// TIA Portal project "Traffic Contol" (V14)

(* hardware
DEVICE "S7-1200 station_1"  S7-1200 Station
   slot 0: "Rack_0"  S7-1200 Rack  Rack  V1.0
   slot 1: "PLC_1"  CPU 1212C AC/DC/Rly  6ES7 212-1BE40-0XB0  V4.2
DEVICE "S7-1200 station_2"  S7-1200 Station
   slot 0: "Rack_0"  S7-1200 Rack  Rack  V1.0
   slot 1: "PLC_2"  CPU 1212C AC/DC/Rly  6ES7 212-1BE40-0XB0  V4.2
*)

// ===== PLC "PLC_1"  CPU 1212C AC/DC/Rly =====

VAR_GLOBAL   // PLC tag table "Default tag table"
   "Switch_0" AT %I0.0 : Bool;
   "Switch_1" AT %I0.1 : Bool;
   "Switch_2" AT %I0.2 : Bool;
   "Switch_3" AT %I0.3 : Bool;
   "Switch_4" AT %I0.4 : Bool;
   "Switch_5" AT %I0.5 : Bool;
   "Switch_6" AT %I0.6 : Bool;
   "Switch_7" AT %I0.7 : Bool;
   "Green_light_1" AT %Q0.0 : Bool;
   "Yellow_light_1" AT %Q0.1 : Bool;
   "Red_light_1" AT %Q0.2 : Bool;
   "Yellow_light_2" AT %Q0.3 : Bool;
   "Red_light_2" AT %Q0.4 : Bool;
   "Green_light_2" AT %Q0.5 : Bool;
   "Delay_1" AT %M0.0 : Bool;
   "Delay_2" AT %M0.1 : Bool;
   "System_Byte" AT %MB1 : Byte;
   "FirstScan" AT %M1.0 : Bool;
   "DiagStatusUpdate" AT %M1.1 : Bool;
   "AlwaysTRUE" AT %M1.2 : Bool;
   "AlwaysFALSE" AT %M1.3 : Bool;
   "System_Byte(1)" AT %MB1 : Byte;
   "Clock_Byte" AT %MB5 : Byte;
   "Clock_10Hz" AT %M5.0 : Bool;
   "Clock_5Hz" AT %M5.1 : Bool;
   "Clock_2.5Hz" AT %M5.2 : Bool;
   "Clock_2Hz" AT %M5.3 : Bool;
   "Clock_1.25Hz" AT %M5.4 : Bool;
   "Clock_1Hz" AT %M5.5 : Bool;
   "Clock_0.625Hz" AT %M5.6 : Bool;
   "Clock_0.5Hz" AT %M5.7 : Bool;
   "ERR" AT %MW2 : Int;
END_VAR

DATA_BLOCK "HOLD_REG"   // DB10
{ S7_Optimized_Access := 'FALSE' }
VERSION : 0.1
   VAR
      BUFFER : Array[0..15] of Bool;
      BUFFER1 : Array[0..15] of Bool;
      FILLER : Array[0..15] of Word;
   END_VAR
BEGIN
   BUFFER[2] := false;
   BUFFER[0] := false;
   BUFFER[6] := false;
END_DATA_BLOCK

DATA_BLOCK "CONFIG_PLC_2"   // DB11
{ S7_Optimized_Access := 'TRUE' }
VERSION : 0.1
   VAR
      Server_IP : TCON_IP_v4;
      DISCONNECT : Bool;
      NDR : Bool;
      DR : Bool;
      ERROR : Bool;
      STATUS : Word;
   END_VAR
BEGIN
   Server_IP.InterfaceId := 64;
   Server_IP.LocalPort := 502;
   Server_IP.ID := 16#01;
END_DATA_BLOCK

DATA_BLOCK "CONFIG_Train"   // DB14
{ S7_Optimized_Access := 'TRUE' }
VERSION : 0.1
   VAR
      Server_IP : TCON_IP_v4;
      DISCONNECT : Bool;
      NDR : Bool;
      DR : Bool;
      ERROR : Bool;
      STATUS : Word;
   END_VAR
BEGIN
   Server_IP.InterfaceId := 64;
   Server_IP.LocalPort := 503;
   Server_IP.ID := 16#03;
END_DATA_BLOCK

DATA_BLOCK "CONFIG_Overide"   // DB15
{ S7_Optimized_Access := 'TRUE' }
VERSION : 0.1
   VAR
      Server_IP : TCON_IP_v4;
      DISCONNECT : Bool := false;
      NDR : Bool := false;
      DR : Bool := false;
      ERROR : Bool := false;
      STATUS : Word := 16#0;
   END_VAR
BEGIN
   Server_IP.InterfaceId := 64;
   Server_IP.LocalPort := 504;
   Server_IP.ID := 16#04;
END_DATA_BLOCK

// folder: System blocks/Program resources

DATA_BLOCK "IEC_Timer_0_DB"   // DB1
{ S7_Optimized_Access := 'TRUE' }
AUTHOR : Simatic
FAMILY : IEC
NAME : IEC_TMR
VERSION : 1.0
// stored: InstanceOfName IEC_TIMER
"IEC_TIMER"
BEGIN
END_DATA_BLOCK

DATA_BLOCK "IEC_Timer_0_DB_1"   // DB2
{ S7_Optimized_Access := 'TRUE' }
AUTHOR : Simatic
FAMILY : IEC
NAME : IEC_TMR
VERSION : 1.0
// stored: InstanceOfName IEC_TIMER
"IEC_TIMER"
BEGIN
END_DATA_BLOCK

DATA_BLOCK "IEC_Timer_0_DB_2"   // DB3
{ S7_Optimized_Access := 'TRUE' }
AUTHOR : Simatic
FAMILY : IEC
NAME : IEC_TMR
VERSION : 1.0
// stored: InstanceOfName IEC_TIMER
"IEC_TIMER"
BEGIN
END_DATA_BLOCK

DATA_BLOCK "IEC_Timer_0_DB_3"   // DB4
{ S7_Optimized_Access := 'TRUE' }
AUTHOR : Simatic
FAMILY : IEC
NAME : IEC_TMR
VERSION : 1.0
// stored: InstanceOfName IEC_TIMER
"IEC_TIMER"
BEGIN
END_DATA_BLOCK

DATA_BLOCK "IEC_Timer_0_DB_4"   // DB5
{ S7_Optimized_Access := 'TRUE' }
AUTHOR : Simatic
FAMILY : IEC
NAME : IEC_TMR
VERSION : 1.0
// stored: InstanceOfName IEC_TIMER
"IEC_TIMER"
BEGIN
END_DATA_BLOCK

DATA_BLOCK "IEC_Timer_0_DB_5"   // DB6
{ S7_Optimized_Access := 'TRUE' }
AUTHOR : Simatic
FAMILY : IEC
NAME : IEC_TMR
VERSION : 1.0
// stored: InstanceOfName IEC_TIMER
"IEC_TIMER"
BEGIN
END_DATA_BLOCK

DATA_BLOCK "IEC_Timer_0_DB_6"   // DB7
{ S7_Optimized_Access := 'TRUE' }
AUTHOR : Simatic
FAMILY : IEC
NAME : IEC_TMR
VERSION : 1.0
// stored: InstanceOfName IEC_TIMER
"IEC_TIMER"
BEGIN
END_DATA_BLOCK

DATA_BLOCK "IEC_Timer_0_DB_7"   // DB8
{ S7_Optimized_Access := 'TRUE' }
AUTHOR : Simatic
FAMILY : IEC
NAME : IEC_TMR
VERSION : 1.0
// stored: InstanceOfName IEC_TIMER
"IEC_TIMER"
BEGIN
END_DATA_BLOCK

DATA_BLOCK "IEC_Timer_0_DB_8"   // DB9
{ S7_Optimized_Access := 'TRUE' }
AUTHOR : Simatic
FAMILY : IEC
NAME : IEC_TMR
VERSION : 1.0
// stored: InstanceOfName IEC_TIMER
"IEC_TIMER"
BEGIN
END_DATA_BLOCK

// folder: (top level)

FUNCTION "Trash" : Void   // FC1, LAD
{ S7_Optimized_Access := 'TRUE' }
VERSION : 0.1
   VAR_TEMP   // added for the SCL form of the ladder/FBD networks
      _w1 : Bool;
   END_VAR
BEGIN

REGION Network 2
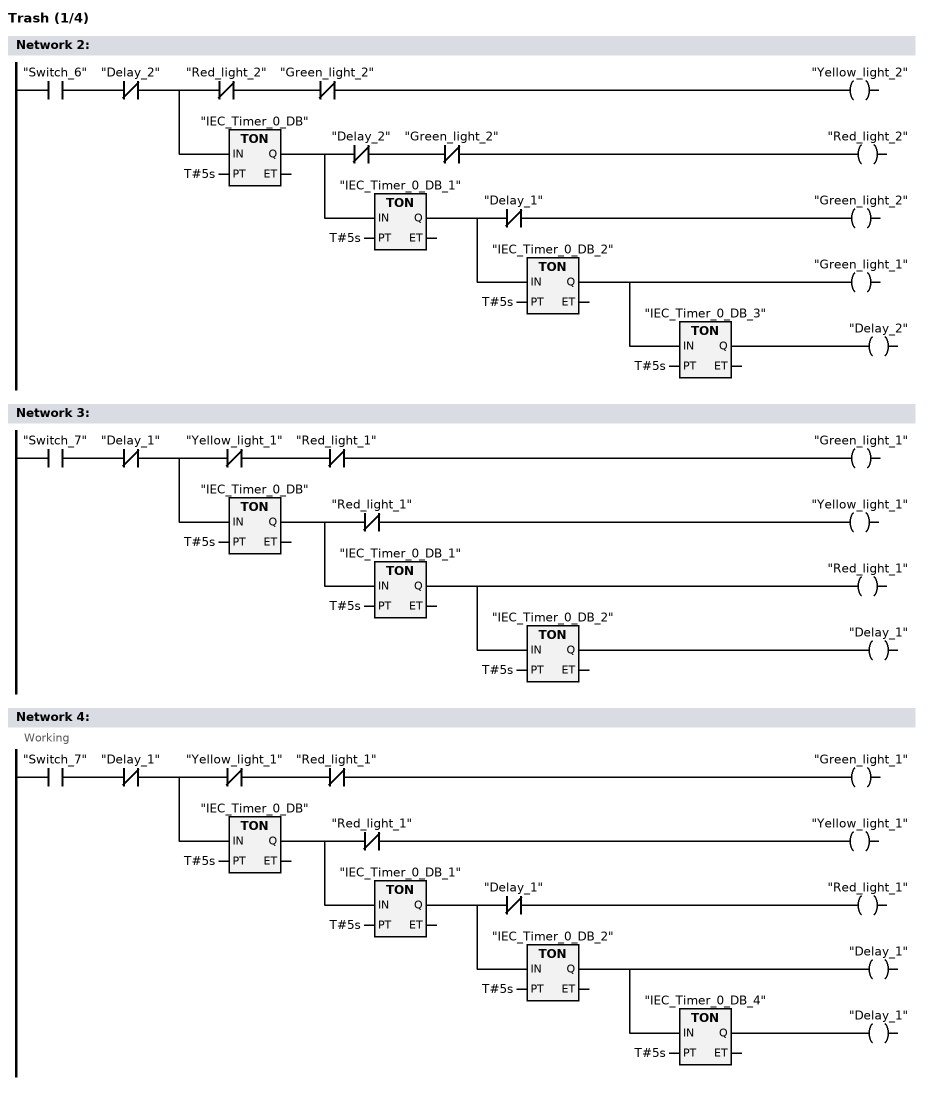
   #_w1 := "Switch_6" AND NOT "Delay_2";
   "Yellow_light_2" := #_w1 AND NOT "Red_light_2" AND NOT "Green_light_2";
   "IEC_Timer_0_DB".TON(IN := #_w1, PT := T#5s);
   "Red_light_2" := "IEC_Timer_0_DB".Q AND NOT "Delay_2" AND NOT "Green_light_2";
   "IEC_Timer_0_DB_1".TON(IN := "IEC_Timer_0_DB".Q, PT := T#5s);
   "Green_light_2" := "IEC_Timer_0_DB_1".Q AND NOT "Delay_1";
   "IEC_Timer_0_DB_2".TON(IN := "IEC_Timer_0_DB_1".Q, PT := T#5s);
   "Green_light_1" := "IEC_Timer_0_DB_2".Q;
   "IEC_Timer_0_DB_3".TON(IN := "IEC_Timer_0_DB_2".Q, PT := T#5s);
   "Delay_2" := "IEC_Timer_0_DB_3".Q;
END_REGION

REGION Network 3
   #_w1 := "Switch_7" AND NOT "Delay_1";
   "Green_light_1" := #_w1 AND NOT "Yellow_light_1" AND NOT "Red_light_1";
   "IEC_Timer_0_DB".TON(IN := #_w1, PT := T#5s);
   "Yellow_light_1" := "IEC_Timer_0_DB".Q AND NOT "Red_light_1";
   "IEC_Timer_0_DB_1".TON(IN := "IEC_Timer_0_DB".Q, PT := T#5s);
   "Red_light_1" := "IEC_Timer_0_DB_1".Q;
   "IEC_Timer_0_DB_2".TON(IN := "IEC_Timer_0_DB_1".Q, PT := T#5s);
   "Delay_1" := "IEC_Timer_0_DB_2".Q;
END_REGION

REGION Network 4
   // Working
   #_w1 := "Switch_7" AND NOT "Delay_1";
   "Green_light_1" := #_w1 AND NOT "Yellow_light_1" AND NOT "Red_light_1";
   "IEC_Timer_0_DB".TON(IN := #_w1, PT := T#5s);
   "Yellow_light_1" := "IEC_Timer_0_DB".Q AND NOT "Red_light_1";
   "IEC_Timer_0_DB_1".TON(IN := "IEC_Timer_0_DB".Q, PT := T#5s);
   "Red_light_1" := "IEC_Timer_0_DB_1".Q AND NOT "Delay_1";
   "IEC_Timer_0_DB_2".TON(IN := "IEC_Timer_0_DB_1".Q, PT := T#5s);
   "Delay_1" := "IEC_Timer_0_DB_2".Q;
   "IEC_Timer_0_DB_4".TON(IN := "IEC_Timer_0_DB_2".Q, PT := T#5s);
   "Delay_1" := "IEC_Timer_0_DB_4".Q;
END_REGION

REGION Network 5
   // Working 123
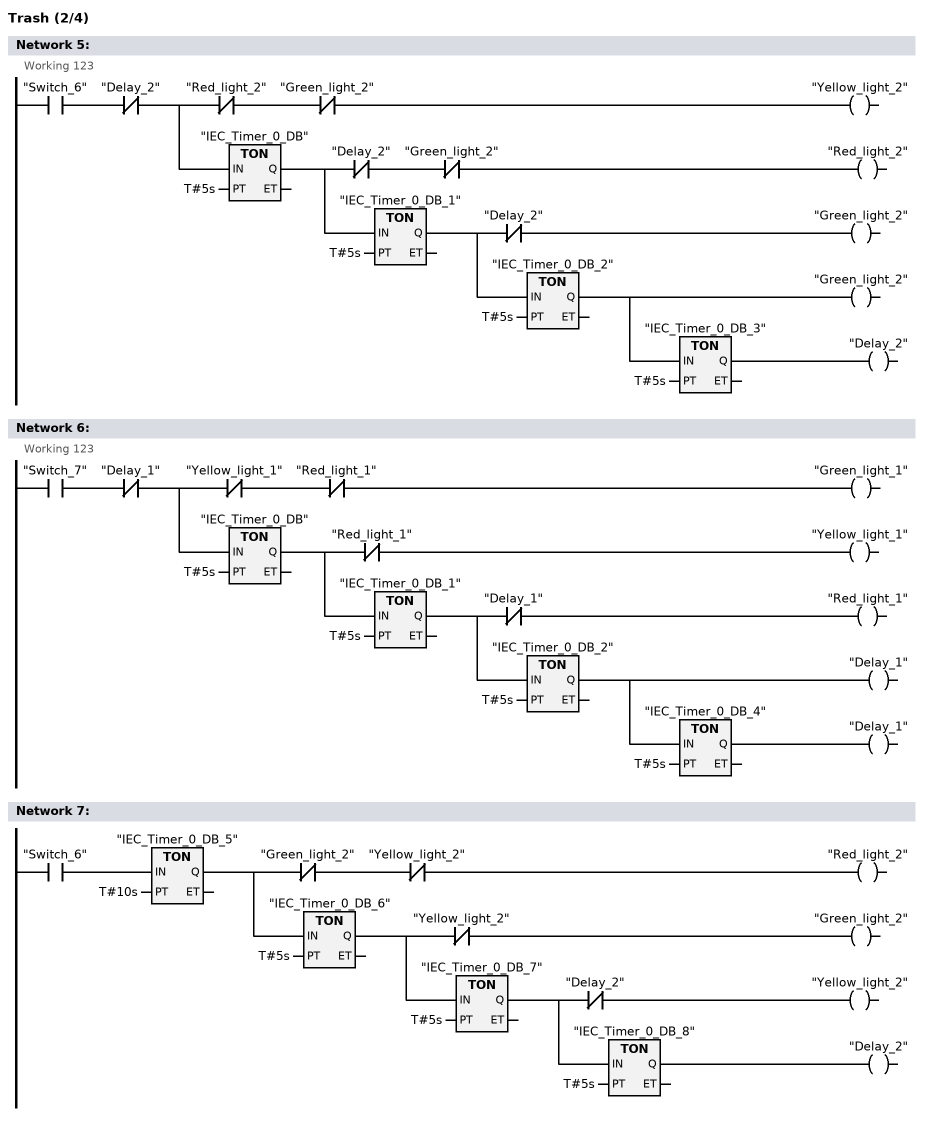
   #_w1 := "Switch_6" AND NOT "Delay_2";
   "Yellow_light_2" := #_w1 AND NOT "Red_light_2" AND NOT "Green_light_2";
   "IEC_Timer_0_DB".TON(IN := #_w1, PT := T#5s);
   "Red_light_2" := "IEC_Timer_0_DB".Q AND NOT "Delay_2" AND NOT "Green_light_2";
   "IEC_Timer_0_DB_1".TON(IN := "IEC_Timer_0_DB".Q, PT := T#5s);
   "Green_light_2" := "IEC_Timer_0_DB_1".Q AND NOT "Delay_2";
   "IEC_Timer_0_DB_2".TON(IN := "IEC_Timer_0_DB_1".Q, PT := T#5s);
   "Green_light_2" := "IEC_Timer_0_DB_2".Q;
   "IEC_Timer_0_DB_3".TON(IN := "IEC_Timer_0_DB_2".Q, PT := T#5s);
   "Delay_2" := "IEC_Timer_0_DB_3".Q;
END_REGION

REGION Network 6
   // Working 123
   #_w1 := "Switch_7" AND NOT "Delay_1";
   "Green_light_1" := #_w1 AND NOT "Yellow_light_1" AND NOT "Red_light_1";
   "IEC_Timer_0_DB".TON(IN := #_w1, PT := T#5s);
   "Yellow_light_1" := "IEC_Timer_0_DB".Q AND NOT "Red_light_1";
   "IEC_Timer_0_DB_1".TON(IN := "IEC_Timer_0_DB".Q, PT := T#5s);
   "Red_light_1" := "IEC_Timer_0_DB_1".Q AND NOT "Delay_1";
   "IEC_Timer_0_DB_2".TON(IN := "IEC_Timer_0_DB_1".Q, PT := T#5s);
   "Delay_1" := "IEC_Timer_0_DB_2".Q;
   "IEC_Timer_0_DB_4".TON(IN := "IEC_Timer_0_DB_2".Q, PT := T#5s);
   "Delay_1" := "IEC_Timer_0_DB_4".Q;
END_REGION

REGION Network 7
   "IEC_Timer_0_DB_5".TON(IN := "Switch_6", PT := T#10s);
   "Red_light_2" := "IEC_Timer_0_DB_5".Q AND NOT "Green_light_2" AND NOT "Yellow_light_2";
   "IEC_Timer_0_DB_6".TON(IN := "IEC_Timer_0_DB_5".Q, PT := T#5s);
   "Green_light_2" := "IEC_Timer_0_DB_6".Q AND NOT "Yellow_light_2";
   "IEC_Timer_0_DB_7".TON(IN := "IEC_Timer_0_DB_6".Q, PT := T#5s);
   "Yellow_light_2" := "IEC_Timer_0_DB_7".Q AND NOT "Delay_2";
   "IEC_Timer_0_DB_8".TON(IN := "IEC_Timer_0_DB_7".Q, PT := T#5s);
   "Delay_2" := "IEC_Timer_0_DB_8".Q;
END_REGION

REGION Network 8
   // working set
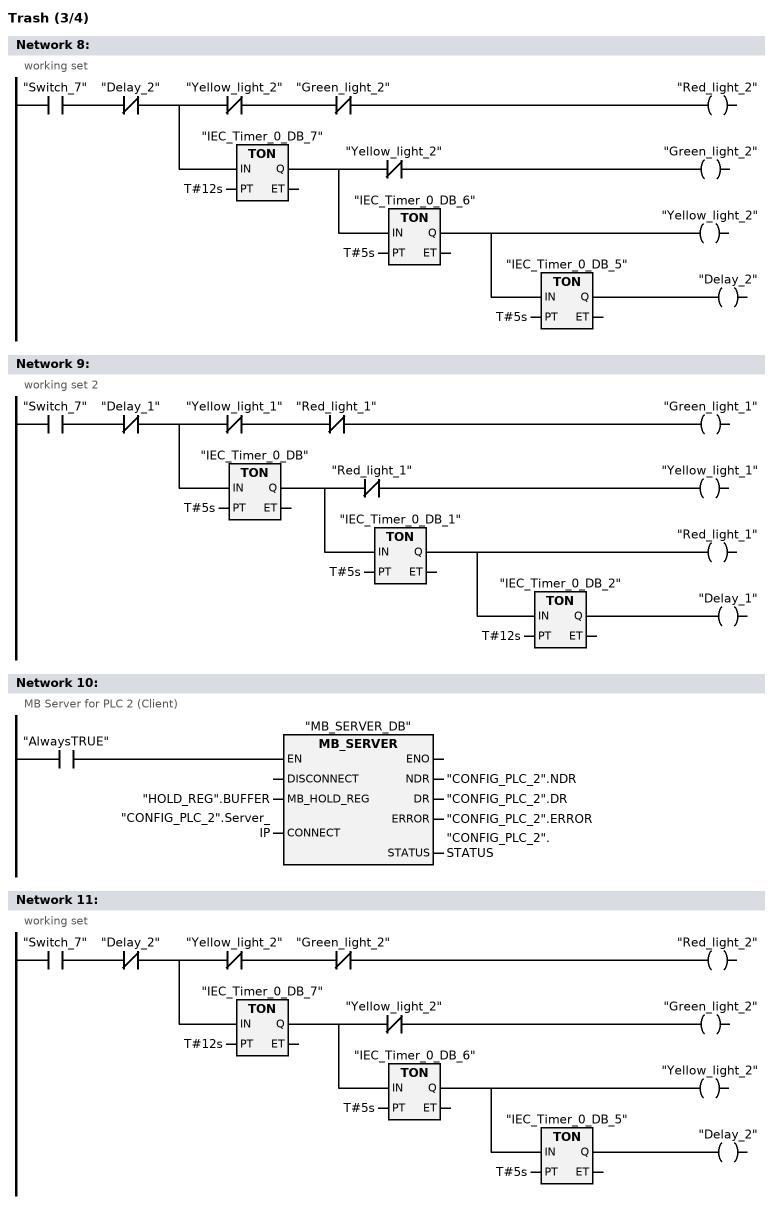
   #_w1 := "Switch_7" AND NOT "Delay_2";
   "Red_light_2" := #_w1 AND NOT "Yellow_light_2" AND NOT "Green_light_2";
   "IEC_Timer_0_DB_7".TON(IN := #_w1, PT := T#12s);
   "Green_light_2" := "IEC_Timer_0_DB_7".Q AND NOT "Yellow_light_2";
   "IEC_Timer_0_DB_6".TON(IN := "IEC_Timer_0_DB_7".Q, PT := T#5s);
   "Yellow_light_2" := "IEC_Timer_0_DB_6".Q;
   "IEC_Timer_0_DB_5".TON(IN := "IEC_Timer_0_DB_6".Q, PT := T#5s);
   "Delay_2" := "IEC_Timer_0_DB_5".Q;
END_REGION

REGION Network 9
   // working set 2
   #_w1 := "Switch_7" AND NOT "Delay_1";
   "Green_light_1" := #_w1 AND NOT "Yellow_light_1" AND NOT "Red_light_1";
   "IEC_Timer_0_DB".TON(IN := #_w1, PT := T#5s);
   "Yellow_light_1" := "IEC_Timer_0_DB".Q AND NOT "Red_light_1";
   "IEC_Timer_0_DB_1".TON(IN := "IEC_Timer_0_DB".Q, PT := T#5s);
   "Red_light_1" := "IEC_Timer_0_DB_1".Q;
   "IEC_Timer_0_DB_2".TON(IN := "IEC_Timer_0_DB_1".Q, PT := T#12s);
   "Delay_1" := "IEC_Timer_0_DB_2".Q;
END_REGION

REGION Network 10
   // MB Server for PLC 2 (Client)
   IF "AlwaysTRUE" THEN
       "MB_SERVER_DB"(MB_HOLD_REG := "HOLD_REG".BUFFER,   // MB_SERVER
                      CONNECT := "CONFIG_PLC_2".Server_IP,
                      NDR => "CONFIG_PLC_2".NDR,
                      DR => "CONFIG_PLC_2".DR,
                      ERROR => "CONFIG_PLC_2".ERROR,
                      STATUS => "CONFIG_PLC_2".STATUS);
   END_IF;
END_REGION

REGION Network 11
   // working set
   #_w1 := "Switch_7" AND NOT "Delay_2";
   "Red_light_2" := #_w1 AND NOT "Yellow_light_2" AND NOT "Green_light_2";
   "IEC_Timer_0_DB_7".TON(IN := #_w1, PT := T#12s);
   "Green_light_2" := "IEC_Timer_0_DB_7".Q AND NOT "Yellow_light_2";
   "IEC_Timer_0_DB_6".TON(IN := "IEC_Timer_0_DB_7".Q, PT := T#5s);
   "Yellow_light_2" := "IEC_Timer_0_DB_6".Q;
   "IEC_Timer_0_DB_5".TON(IN := "IEC_Timer_0_DB_6".Q, PT := T#5s);
   "Delay_2" := "IEC_Timer_0_DB_5".Q;
END_REGION

REGION Network 12
   // working set 2
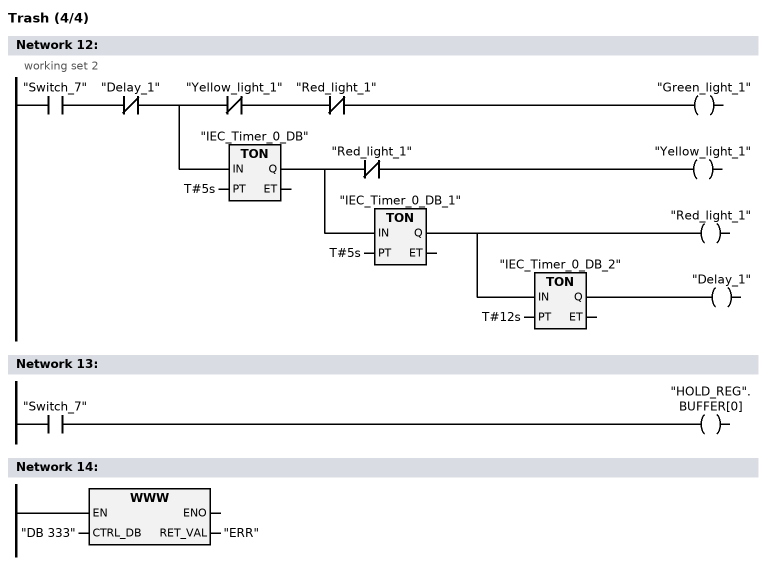
   #_w1 := "Switch_7" AND NOT "Delay_1";
   "Green_light_1" := #_w1 AND NOT "Yellow_light_1" AND NOT "Red_light_1";
   "IEC_Timer_0_DB".TON(IN := #_w1, PT := T#5s);
   "Yellow_light_1" := "IEC_Timer_0_DB".Q AND NOT "Red_light_1";
   "IEC_Timer_0_DB_1".TON(IN := "IEC_Timer_0_DB".Q, PT := T#5s);
   "Red_light_1" := "IEC_Timer_0_DB_1".Q;
   "IEC_Timer_0_DB_2".TON(IN := "IEC_Timer_0_DB_1".Q, PT := T#12s);
   "Delay_1" := "IEC_Timer_0_DB_2".Q;
END_REGION

REGION Network 13
   RUNG wire#powerrail
      Contact( "Switch_7" )
      Coil( "HOLD_REG".BUFFER[0] )
   END_RUNG
   // the same network as SCL:
   "HOLD_REG".BUFFER[0] := "Switch_7";
END_REGION

REGION Network 14
   "ERR" := WWW(CTRL_DB := "DB 333");
END_REGION
END_FUNCTION

ORGANIZATION_BLOCK "Main"   // OB1, LAD, ProgramCycle
TITLE = "Main Program Sweep (Cycle)"
{ S7_Optimized_Access := 'TRUE' }
VERSION : 0.1
   VAR_INPUT
      Initial_Call : Bool;   // Initial call of this OB
      Remanence : Bool;   // =True, if remanent data are available
   END_VAR
   VAR_TEMP   // added for the SCL form of the ladder/FBD networks
      _w1 : Bool;
   END_VAR
BEGIN

REGION Network 1
   // MB Server for overide
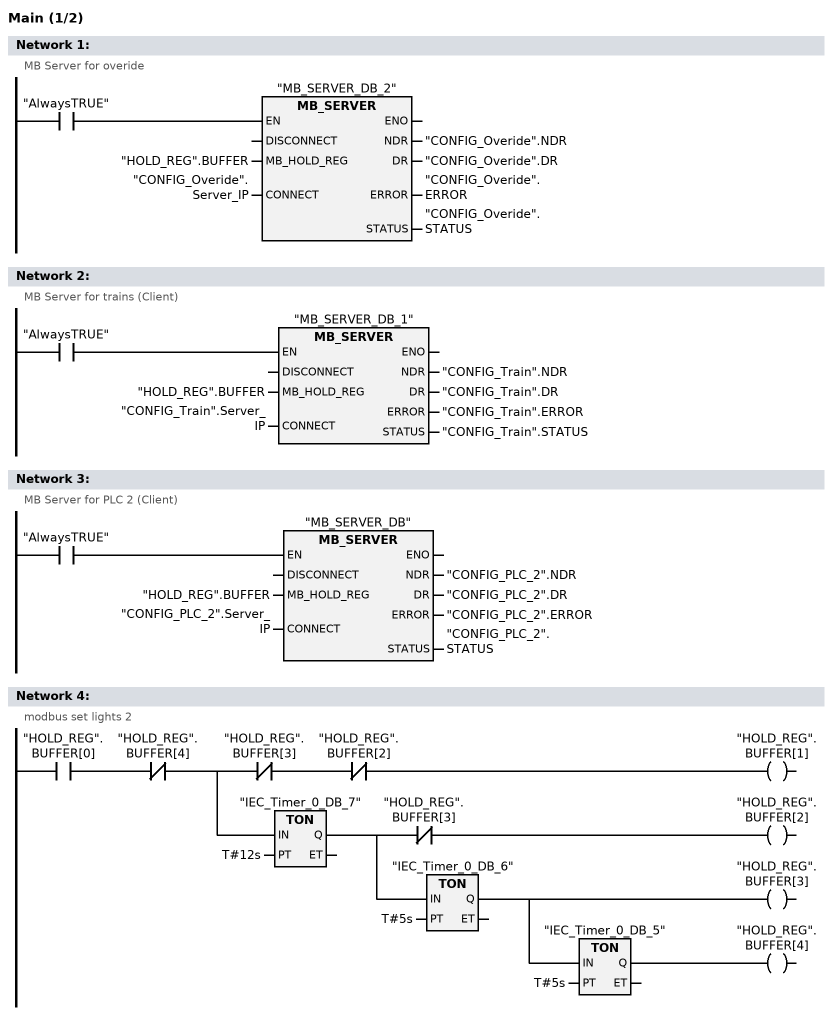
   IF "AlwaysTRUE" THEN
       "MB_SERVER_DB_2"(MB_HOLD_REG := "HOLD_REG".BUFFER,   // MB_SERVER
                        CONNECT := "CONFIG_Overide".Server_IP,
                        NDR => "CONFIG_Overide".NDR,
                        DR => "CONFIG_Overide".DR,
                        ERROR => "CONFIG_Overide".ERROR,
                        STATUS => "CONFIG_Overide".STATUS);
   END_IF;
END_REGION

REGION Network 2
   // MB Server for trains (Client)
   IF "AlwaysTRUE" THEN
       "MB_SERVER_DB_1"(MB_HOLD_REG := "HOLD_REG".BUFFER,   // MB_SERVER
                        CONNECT := "CONFIG_Train".Server_IP,
                        NDR => "CONFIG_Train".NDR,
                        DR => "CONFIG_Train".DR,
                        ERROR => "CONFIG_Train".ERROR,
                        STATUS => "CONFIG_Train".STATUS);
   END_IF;
END_REGION

REGION Network 3
   // MB Server for PLC 2 (Client)
   IF "AlwaysTRUE" THEN
       "MB_SERVER_DB"(MB_HOLD_REG := "HOLD_REG".BUFFER,   // MB_SERVER
                      CONNECT := "CONFIG_PLC_2".Server_IP,
                      NDR => "CONFIG_PLC_2".NDR,
                      DR => "CONFIG_PLC_2".DR,
                      ERROR => "CONFIG_PLC_2".ERROR,
                      STATUS => "CONFIG_PLC_2".STATUS);
   END_IF;
END_REGION

REGION Network 4
   // modbus set lights 2
   #_w1 := "HOLD_REG".BUFFER[0] AND NOT "HOLD_REG".BUFFER[4];
   "HOLD_REG".BUFFER[1] := #_w1 AND NOT "HOLD_REG".BUFFER[3] AND NOT "HOLD_REG".BUFFER[2];
   "IEC_Timer_0_DB_7".TON(IN := #_w1, PT := T#12s);
   "HOLD_REG".BUFFER[2] := "IEC_Timer_0_DB_7".Q AND NOT "HOLD_REG".BUFFER[3];
   "IEC_Timer_0_DB_6".TON(IN := "IEC_Timer_0_DB_7".Q, PT := T#5s);
   "HOLD_REG".BUFFER[3] := "IEC_Timer_0_DB_6".Q;
   "IEC_Timer_0_DB_5".TON(IN := "IEC_Timer_0_DB_6".Q, PT := T#5s);
   "HOLD_REG".BUFFER[4] := "IEC_Timer_0_DB_5".Q;
END_REGION

REGION Network 5
   // modbus set lights 1
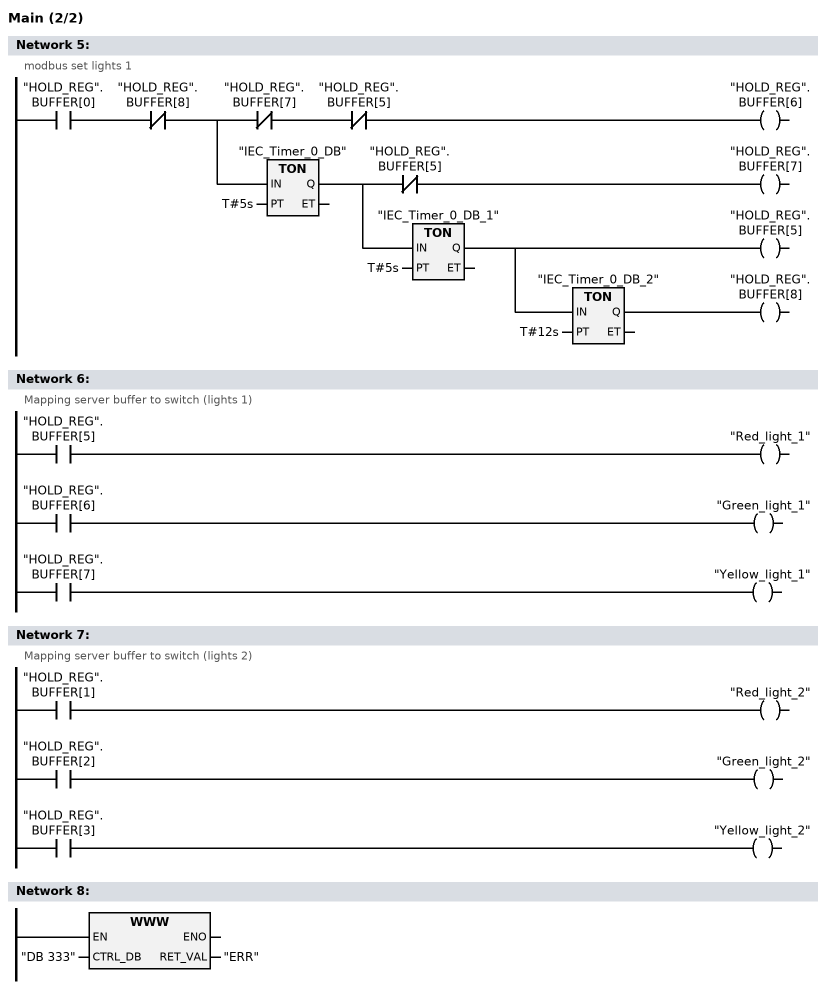
   #_w1 := "HOLD_REG".BUFFER[0] AND NOT "HOLD_REG".BUFFER[8];
   "HOLD_REG".BUFFER[6] := #_w1 AND NOT "HOLD_REG".BUFFER[7] AND NOT "HOLD_REG".BUFFER[5];
   "IEC_Timer_0_DB".TON(IN := #_w1, PT := T#5s);
   "HOLD_REG".BUFFER[7] := "IEC_Timer_0_DB".Q AND NOT "HOLD_REG".BUFFER[5];
   "IEC_Timer_0_DB_1".TON(IN := "IEC_Timer_0_DB".Q, PT := T#5s);
   "HOLD_REG".BUFFER[5] := "IEC_Timer_0_DB_1".Q;
   "IEC_Timer_0_DB_2".TON(IN := "IEC_Timer_0_DB_1".Q, PT := T#12s);
   "HOLD_REG".BUFFER[8] := "IEC_Timer_0_DB_2".Q;
END_REGION

REGION Network 6
   // Mapping server buffer to switch (lights 1)
   RUNG wire#powerrail
      Contact( "HOLD_REG".BUFFER[5] )
      Coil( "Red_light_1" )
   END_RUNG
   RUNG wire#powerrail
      Contact( "HOLD_REG".BUFFER[6] )
      Coil( "Green_light_1" )
   END_RUNG
   RUNG wire#powerrail
      Contact( "HOLD_REG".BUFFER[7] )
      Coil( "Yellow_light_1" )
   END_RUNG
   // the same network as SCL:
   "Red_light_1" := "HOLD_REG".BUFFER[5];
   "Green_light_1" := "HOLD_REG".BUFFER[6];
   "Yellow_light_1" := "HOLD_REG".BUFFER[7];
END_REGION

REGION Network 7
   // Mapping server buffer to switch (lights 2)
   RUNG wire#powerrail
      Contact( "HOLD_REG".BUFFER[1] )
      Coil( "Red_light_2" )
   END_RUNG
   RUNG wire#powerrail
      Contact( "HOLD_REG".BUFFER[2] )
      Coil( "Green_light_2" )
   END_RUNG
   RUNG wire#powerrail
      Contact( "HOLD_REG".BUFFER[3] )
      Coil( "Yellow_light_2" )
   END_RUNG
   // the same network as SCL:
   "Red_light_2" := "HOLD_REG".BUFFER[1];
   "Green_light_2" := "HOLD_REG".BUFFER[2];
   "Yellow_light_2" := "HOLD_REG".BUFFER[3];
END_REGION

REGION Network 8
   "ERR" := WWW(CTRL_DB := "DB 333");
END_REGION
END_ORGANIZATION_BLOCK

// ===== PLC "PLC_2"  CPU 1212C AC/DC/Rly =====

VAR_GLOBAL   // PLC tag table "Default tag table"
   "System_Byte" AT %MB1 : Byte;
   "FirstScan" AT %M1.0 : Bool;
   "DiagStatusUpdate" AT %M1.1 : Bool;
   "AlwaysTRUE" AT %M1.2 : Bool;
   "AlwaysFALSE" AT %M1.3 : Bool;
   "Clock_Byte" AT %MB5 : Byte;
   "Clock_10Hz" AT %M5.0 : Bool;
   "Clock_5Hz" AT %M5.1 : Bool;
   "Clock_2.5Hz" AT %M5.2 : Bool;
   "Clock_2Hz" AT %M5.3 : Bool;
   "Clock_1.25Hz" AT %M5.4 : Bool;
   "Clock_1Hz" AT %M5.5 : Bool;
   "Clock_0.625Hz" AT %M5.6 : Bool;
   "Clock_0.5Hz" AT %M5.7 : Bool;
END_VAR

VAR_GLOBAL   // PLC tag table "Traffic Tag"
   "Switch_0" AT %I0.0 : Bool;
   "Switch_1" AT %I0.1 : Bool;
   "Switch_2" AT %I0.2 : Bool;
   "Switch_3" AT %I0.3 : Bool;
   "Switch_4" AT %I0.4 : Bool;
   "Switch_5" AT %I0.5 : Bool;
   "Switch_6" AT %I0.6 : Bool;
   "Switch_7" AT %I0.7 : Bool;
   "Green_light_1" AT %Q0.0 : Bool;
   "Yellow_light_1" AT %Q0.1 : Bool;
   "Red_light_1" AT %Q0.2 : Bool;
   "Yellow_light_2" AT %Q0.3 : Bool;
   "Red_light_2" AT %Q0.4 : Bool;
   "Green_light_2" AT %Q0.5 : Bool;
   "Delay_1" AT %M0.0 : Bool;
   "Delay_2" AT %M0.1 : Bool;
END_VAR

DATA_BLOCK "CLIENT_CONFIG"   // DB2
{ S7_Optimized_Access := 'TRUE' }
VERSION : 0.1
   VAR
      Server_IP : TCON_IP_v4;
      DISCONNECT : Bool;
      DONE : Bool;
      BUSY : Bool;
      ERROR : Bool;
      STATUS : Word;
   END_VAR
BEGIN
   Server_IP.ID := 16#02;
   Server_IP.ActiveEstablished := 1;
   Server_IP.RemoteAddress.ADDR[1] := 16#0A;
   Server_IP.RemoteAddress.ADDR[2] := 16#0A;
   Server_IP.RemoteAddress.ADDR[3] := 16#1E;
   Server_IP.RemoteAddress.ADDR[4] := 16#02;
   Server_IP.RemotePort := 502;
   Server_IP.InterfaceId := 64;
END_DATA_BLOCK

DATA_BLOCK "HOLD_REG_PTR"   // DB10
{ S7_Optimized_Access := 'FALSE' }
VERSION : 0.1
   VAR
      BUFFER : Array[0..15] of Bool;
      BUFFER1 : Array[0..15] of Bool;
   END_VAR
BEGIN
END_DATA_BLOCK

FUNCTION "Trash" : Void   // FC1, LAD
{ S7_Optimized_Access := 'TRUE' }
VERSION : 0.1
BEGIN

REGION Network 2
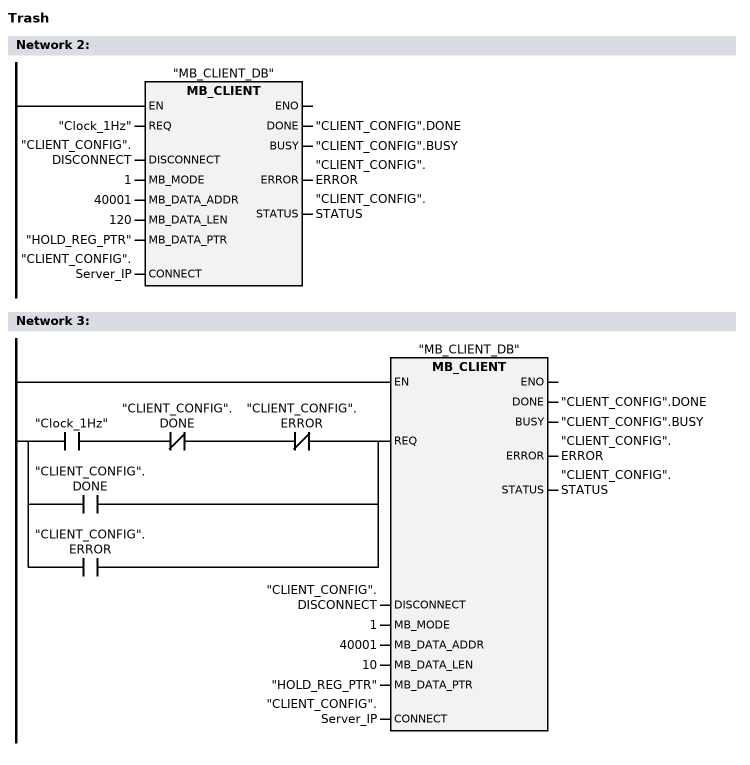
   "MB_CLIENT_DB"(REQ := "Clock_1Hz",   // MB_CLIENT
                  DISCONNECT := "CLIENT_CONFIG".DISCONNECT,
                  MB_MODE := 1,
                  MB_DATA_ADDR := 40001,
                  MB_DATA_LEN := 120,
                  MB_DATA_PTR := "HOLD_REG_PTR",
                  CONNECT := "CLIENT_CONFIG".Server_IP,
                  DONE => "CLIENT_CONFIG".DONE,
                  BUSY => "CLIENT_CONFIG".BUSY,
                  ERROR => "CLIENT_CONFIG".ERROR,
                  STATUS => "CLIENT_CONFIG".STATUS);
END_REGION

REGION Network 3
   "MB_CLIENT_DB"(REQ := ("Clock_1Hz" AND NOT "CLIENT_CONFIG".DONE AND NOT "CLIENT_CONFIG".ERROR) OR "CLIENT_CONFIG".DONE OR "CLIENT_CONFIG".ERROR,   // MB_CLIENT
                  DISCONNECT := "CLIENT_CONFIG".DISCONNECT,
                  MB_MODE := 1,
                  MB_DATA_ADDR := 40001,
                  MB_DATA_LEN := 10,
                  MB_DATA_PTR := "HOLD_REG_PTR",
                  CONNECT := "CLIENT_CONFIG".Server_IP,
                  DONE => "CLIENT_CONFIG".DONE,
                  BUSY => "CLIENT_CONFIG".BUSY,
                  ERROR => "CLIENT_CONFIG".ERROR,
                  STATUS => "CLIENT_CONFIG".STATUS);
END_REGION
END_FUNCTION

ORGANIZATION_BLOCK "Main"   // OB1, LAD, ProgramCycle
TITLE = "Main Program Sweep (Cycle)"
{ S7_Optimized_Access := 'TRUE' }
VERSION : 0.1
   VAR_INPUT
      Initial_Call : Bool;   // Initial call of this OB
      Remanence : Bool;   // =True, if remanent data are available
   END_VAR
BEGIN

REGION Network 1
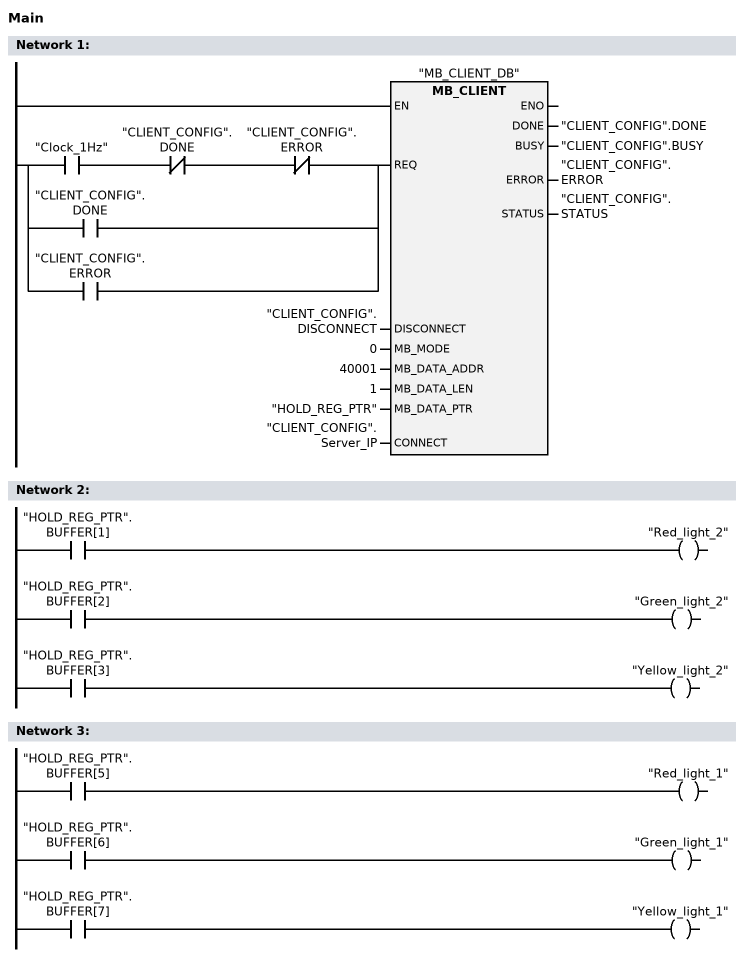
   "MB_CLIENT_DB"(REQ := ("Clock_1Hz" AND NOT "CLIENT_CONFIG".DONE AND NOT "CLIENT_CONFIG".ERROR) OR "CLIENT_CONFIG".DONE OR "CLIENT_CONFIG".ERROR,   // MB_CLIENT
                  DISCONNECT := "CLIENT_CONFIG".DISCONNECT,
                  MB_MODE := 0,
                  MB_DATA_ADDR := 40001,
                  MB_DATA_LEN := 1,
                  MB_DATA_PTR := "HOLD_REG_PTR",
                  CONNECT := "CLIENT_CONFIG".Server_IP,
                  DONE => "CLIENT_CONFIG".DONE,
                  BUSY => "CLIENT_CONFIG".BUSY,
                  ERROR => "CLIENT_CONFIG".ERROR,
                  STATUS => "CLIENT_CONFIG".STATUS);
END_REGION

REGION Network 2
   RUNG wire#powerrail
      Contact( "HOLD_REG_PTR".BUFFER[1] )
      Coil( "Red_light_2" )
   END_RUNG
   RUNG wire#powerrail
      Contact( "HOLD_REG_PTR".BUFFER[2] )
      Coil( "Green_light_2" )
   END_RUNG
   RUNG wire#powerrail
      Contact( "HOLD_REG_PTR".BUFFER[3] )
      Coil( "Yellow_light_2" )
   END_RUNG
   // the same network as SCL:
   "Red_light_2" := "HOLD_REG_PTR".BUFFER[1];
   "Green_light_2" := "HOLD_REG_PTR".BUFFER[2];
   "Yellow_light_2" := "HOLD_REG_PTR".BUFFER[3];
END_REGION

REGION Network 3
   RUNG wire#powerrail
      Contact( "HOLD_REG_PTR".BUFFER[5] )
      Coil( "Red_light_1" )
   END_RUNG
   RUNG wire#powerrail
      Contact( "HOLD_REG_PTR".BUFFER[6] )
      Coil( "Green_light_1" )
   END_RUNG
   RUNG wire#powerrail
      Contact( "HOLD_REG_PTR".BUFFER[7] )
      Coil( "Yellow_light_1" )
   END_RUNG
   // the same network as SCL:
   "Red_light_1" := "HOLD_REG_PTR".BUFFER[5];
   "Green_light_1" := "HOLD_REG_PTR".BUFFER[6];
   "Yellow_light_1" := "HOLD_REG_PTR".BUFFER[7];
END_REGION
END_ORGANIZATION_BLOCK